// TwinCAT 3 PLC project main
// ProgramVersion: 3.1.4024.0
// libraries:
//   Tc2_Math, * (Beckhoff Automation GmbH)
//   Tc2_Standard, * (Beckhoff Automation GmbH)
//   Tc2_System, * (Beckhoff Automation GmbH)
//   Tc3_Module, * (Beckhoff Automation GmbH)
//   Title,2.0,HSLU
// project tree:
//   DUTs/ PID_Parameter_Strukt.TcDUT, PT1T2_Parameter_Strukt.TcDUT, System_Modus_Enum.TcDUT
//   / PlcTask.TcTTO
//   POUs/ MAIN.TcPOU, PID_Regler.TcPOU, PT1T2_Prozess.TcPOU
// real-time tasks:
//   TASK PlcTask: cycle T#1ms, priority 20, ADS port 350

CONFIGURATION main
    RESOURCE PLC ON TwinCAT3
        TASK PlcTask(INTERVAL := T#1ms, PRIORITY := 20);
        PROGRAM MAIN WITH PlcTask : MAIN;
    END_RESOURCE
END_CONFIGURATION

// ---- DUTs/PID_Parameter_Strukt.TcDUT
TYPE PID_Parameter_Strukt :
STRUCT
	Kp :		REAL;
	Ti :		REAL;
	Td :		REAL;
	N :			REAL;
	ARW :		BOOL;
	Tr :		REAL;
	umin :		REAL;
	umax :		REAL;
END_STRUCT
END_TYPE

// ---- DUTs/PT1T2_Parameter_Strukt.TcDUT
TYPE PT1T2_Parameter_Strukt :
STRUCT
	K :			REAL;
	T1 :		REAL;
	T2 :		REAL;
END_STRUCT
END_TYPE

// ---- DUTs/System_Modus_Enum.TcDUT
{attribute 'qualified_only'}
{attribute 'strict'}
TYPE System_Modus_Enum :
(
	System_Init := 0,
	System_Run
);
END_TYPE

// ---- POUs/MAIN.TcPOU
PROGRAM MAIN
VAR
	PT1T2Parameter :			PT1T2_Parameter_Strukt;
	PID_Parameter :				PID_Parameter_Strukt;
	Modus :						System_Modus_Enum := System_Modus_Enum.System_Init;
	T :							REAL := 0.001;
	PID_1 :						PID_Regler;
	PT1T2_1 :					PT1T2_Prozess;
	r0 :						REAL := 0;	
	e0 :						REAL := 0;
	
	t_time: 					REAL := 0;
END_VAR

CASE Modus OF
	System_Modus_Enum.System_Init:
	PT1T2Parameter.K := 10;
	PT1T2Parameter.T1 := 0.1;
	PT1T2Parameter.T2 := 0.01;

	PID_Parameter.Kp := 100/PT1T2Parameter.K;
	PID_Parameter.Ti := PT1T2Parameter.T1;
	PID_Parameter.Td := PT1T2Parameter.T2;
	PID_Parameter.N := 10;
	PID_Parameter.umax := 10;
	PID_Parameter.umin := 0;
	PID_Parameter.ARW := TRUE;
	PID_Parameter.Tr := 0.1;
	PID_1(r1 := r0, y1 := PT1T2_1.y, Modus := Modus, Param := PID_Parameter, T := T);
	PT1T2_1(u := PID_1.u, Modus := Modus, Param := PT1T2Parameter, T := T);
	Modus := System_Modus_Enum.System_Run
	;
	System_Modus_Enum.System_Run:
	r0 := PwmSignal(ymin := 25, ymax:= 75, w:=1, yoff:=0, PWM:= 0.5, t_time);
	e0 := r0 - PT1T2_1.y;
	PID_1(r1 := r0, y1 := PT1T2_1.y, Modus := Modus, Param := PID_Parameter, T := T);
	PT1T2_1(u := PID_1.u, Modus := Modus, Param := PT1T2Parameter, T := T);
	t_time := t_time + T;
	;
END_CASE

END_PROGRAM

// ---- POUs/PID_Regler.TcPOU
FUNCTION_BLOCK PID_Regler
VAR_INPUT
	r1 :			REAL;
	y1 :			REAL;
	Modus :		System_Modus_Enum;
	Param :		PID_Parameter_Strukt;
	T :			REAL;
END_VAR
VAR_OUTPUT
	u :			REAL;
END_VAR
VAR
	a0 :		REAL;
	b0 :		REAL;
	c0 :		REAL;

	rm :		REAL;
	ym :		REAL;
	u_temp :	REAL;
	up : 		REAL;
	ui :		REAL;
	ud :		REAL;
	uim :		REAL;
	udm :		REAL;
END_VAR

CASE Modus OF
	System_Modus_Enum.System_Init:
	c0 := (T*Param.Kp)/(2*Param.Ti);
	a0 := (Param.Td)/(Param.Td+Param.N*T);
	b0 := (Param.Kp*Param.Td*Param.N)/(Param.Td+Param.N*T);
	u := 0;
	rm := 0;
	ym := 0;
	up := 0;
	ui := 0;
	ud := 0;
	uim := 0;
	udm := 0;
	;
	System_Modus_Enum.System_Run:
	up := (r1-y1) * Param.Kp;
	IF Param.ARW = TRUE THEN
		ui := uim + c0*((r1-y1)+(rm-ym)) + (T/Param.Tr)*(u-u_temp);
	ELSE
		ui := uim + c0*((r1-y1)+(rm-ym));
	END_IF
	ud := b0 * ((r1-y1)-(rm-ym)) + a0 * udm;
	u := up + ui + ud;
	u_temp := u;
	IF u >= Param.umax THEN
		u := Param.umax;
	END_IF
	IF u <= Param.umin THEN
		u := Param.umin;
	END_IF
	rm := r1;
	ym := y1;
	uim := ui;
	udm := ud;
	;
END_CASE

END_FUNCTION_BLOCK

// ---- POUs/PT1T2_Prozess.TcPOU
FUNCTION_BLOCK PT1T2_Prozess
VAR_INPUT
	u :			REAL;
	Modus :		System_Modus_Enum;
	Param :		PT1T2_Parameter_Strukt;
	T :			REAL;
END_VAR
VAR_OUTPUT
	y :			REAL;
END_VAR
VAR
	alpha1 :	REAL;
	alpha2 :	REAL;
	a1 :		REAL;
	a2 :		REAL;
	b0 :		REAL;
	b1 :		REAL;
	b2 :		REAL;
	
	ym :		REAL;
	ymm :		REAL;
END_VAR

CASE Modus OF
	System_Modus_Enum.System_Init:
	alpha1 := T + Param.T1;
	alpha2 := T + Param.T2;
	a1 := 1;
	a2 := 2;
	b0 := (Param.K*T*T)/(alpha1*alpha2);
	a1 := -((Param.T1/alpha1)+(Param.T2/alpha2));
	a2 := (Param.T1*Param.T2)/(alpha1*alpha2);
	y := 0;
	ym := 0;
	ymm := 0;
	;
	System_Modus_Enum.System_Run:
	y := -a1 * ym - a2 *ymm + b0 * u;
	ymm := ym;
	ym := y;
	;
END_CASE

END_FUNCTION_BLOCK
